TYPE DUT_SERVER_MODULE_INTERFACE_INPUT :
STRUCT
	///Mode to run (init,auto,manual,..)
	Mode: INT;
	///check if the modules is alive
	ConnectionTestInput: BOOL;
	///Modules get their position
	PositionInput : LREAL;
	///Update data= TRUE, No updatedata=FALSE
	Watchbit: BOOL;
	///Emergency stop
	EmergencyStop: BOOL;
	///Range of INPUT skills
	SkillInput: DUT_SERVER_SKILLINPUTARRAY;
END_STRUCT
END_TYPE

(* stored: Version 1.1.0.1, ProductVersion 3.1.0.25
   DUT DUT_SERVER_MODULE_INTERFACE_INPUT: Id {fda85ace-5e82-4edd-8e3c-7e530c8ef3cd} *)
